// TIA Portal V17 export
// export: Created 2024-09-03T21:54:54.8322856Z, ExportSetting WithDefaults, DisplayName Totally Integrated Automation Portal, DisplayVersion V17 Update 7, DisplayName TIA Portal Openness, DisplayVersion V17 Update 7, DisplayName TIA Portal Version Control Interface, DisplayVersion V17, DisplayName SINAMICS Startdrive Advanced, DisplayVersion V17 SP2, DisplayName SINAMICS Startdrive G110M, G120, G120C, G120D, G120P, G115D, DisplayVersion V17 SP2, DisplayName SINAMICS Startdrive G130, G150, S120, S150, SINAMICS MV, S210, DisplayVersion V17 SP2, DisplayName STEP 7 Professional, DisplayVersion V17 Update 7, DisplayName STEP 7 Safety, DisplayVersion V17 Update 6, DisplayName WinCC Advanced / Unified PC, DisplayVersion V17 Update 7
DATA_BLOCK "DB_ProductionProgramActual"   // DB6101
{ S7_Optimized_Access := 'TRUE' }
VERSION : 0.1
// stored: AutoNumber false, DBAccessibleFromOPCUA true, DBAccessibleFromWebserver true, IsOnlyStoredInLoadMemory false, IsRetainMemResEnabled false, IsWriteProtectedInAS false, MemoryReserve 100
   VAR
      Program { S7_SetPoint := 'True'} : "UDT_ProductionProgram";
      ProgrammNumber { S7_SetPoint := 'True'} : Int := 5;
      Load : Bool := FALSE;
      Save : Bool := FALSE;
      CanBeChanged : Bool := FALSE;
   END_VAR
BEGIN
   Program."Name" := 'startup';
   Program.CupformingParametersLeft.DigiforceProgram := 1;
   Program.CupformingParametersLeft.FinalSpeed := 25.0;
   Program.CupformingParametersLeft.ApproachSpeed := 25.0;
   Program.CupformingParametersLeft.FinalForce := 10.0;
   Program.CupformingParametersLeft.ApproachForce := 10.0;
   Program.CupformingParametersLeft.EndWayImmediate := 2.55;
   Program.CupformingParametersLeft.EndWayWithTimeout := 3.0;
   Program.CupformingParametersLeft.SwitchingWay := 20.0;
   Program.CupformingParametersLeft.EndWayTimeout := T#300MS;
   Program.CupformingParametersRight.DigiforceProgram := 1;
   Program.CupformingParametersRight.FinalSpeed := 25.0;
   Program.CupformingParametersRight.ApproachSpeed := 25.0;
   Program.CupformingParametersRight.FinalForce := 10.0;
   Program.CupformingParametersRight.ApproachForce := 10.0;
   Program.CupformingParametersRight.EndWayImmediate := 2.7;
   Program.CupformingParametersRight.EndWayWithTimeout := 3.0;
   Program.CupformingParametersRight.SwitchingWay := 20.0;
   Program.CupformingParametersRight.EndWayTimeout := T#300MS;
   Program.St1Insertion[1] := TRUE;
   Program.St1Insertion[2] := FALSE;
   Program.St1Insertion[3..5] := TRUE;
   Program.St1Insertion[6] := FALSE;
   Program.St1Insertion[7] := TRUE;
   Program.St1Insertion[8] := FALSE;
   Program.St1Insertion[9..10] := TRUE;
   Program.St1Insertion[11] := FALSE;
   Program.St1Insertion[12..17] := TRUE;
   Program.St1Insertion[18] := FALSE;
   Program.St1Insertion[19] := TRUE;
   Program.St1Insertion[20] := FALSE;
   Program.St1InsertionUsed[1..7] := TRUE;
   Program.St1InsertionUsed[8] := FALSE;
   Program.St1InsertionUsed[9..19] := TRUE;
   Program.St1InsertionUsed[20] := FALSE;
   Program.FaureciaNumber := '2567208X';
   Program.FaureciaNumberStartChar := 9;
   Program.FaureciaNumberLength := 8;
   Program.MechanicalType := 0;
END_DATA_BLOCK
